Universal Robots PolyScope program: TCP Test 01.urp

Program TCP Test 01 (installation=default directory=/programs createdIn=5.9.1.1031110 lastSavedIn=5.9.1.1031110 robotSerialNumber=20195501059)
Calibrated DH parameters: a=[0.000146, -0.418764, -0.053981, 0.000058, -0.000023, 0]; d=[0.162545, 37.319448, -206.067439, 168.881546, 0.09955, 0.099464]; alpha=[1.57004, -0.001979, 0.002304, 1.570607, -1.57066, 0]; deltaTheta=[0, -0.174616, -1.258233, 1.432844, -0.000001, 0]
BeforeStart
  URCap Gripper Activate (Robotiq_Grippers, Robotiq Inc.) dataModel(ResetAndActivateKey=false)
  URCap Gripper (Robotiq_Grippers, Robotiq Inc.) dataModel(position=100.0, force=100.0, speed=100.0, positionInDouble=100.0, forceInDouble=100.0, speedInDouble=100.0, slaveIds=[9], blocking=true)
Robot Program (runOnlyOnce=true)
  '2F85 Tool vertical above box'
  MoveJ speed 60 deg/s, acceleration 80 deg/s^2 (useActiveTCP=false) tcp=TCP_2F85; feature=Base
    Waypoint hover: TCP in base x=299.991 y=-399.96 z=49.999 mm, rx=0.0001 ry=0.0001 rz=0 rad; joints [111.356, -78.636, 119.104, -130.453, 270.052, 201.393] deg; TCP offset x=0 y=0 z=175 mm, rx=3.1416 ry=0 rz=0 rad
    Waypoint on_target: TCP in base x=300.002 y=-399.956 z=0.996 mm, rx=0.0001 ry=0 rz=0 rad; joints [111.352, -73.264, 121.787, -138.509, 270.053, 201.401] deg; TCP offset x=0 y=0 z=175 mm, rx=3.1416 ry=0 rz=0 rad
  MoveJ speed 60 deg/s, acceleration 80 deg/s^2 (useActiveTCP=false) tcp=TCP_Mono; feature=Base
    Waypoint on_target: TCP in base x=300.002 y=-399.956 z=0.996 mm, rx=0.0001 ry=0 rz=0 rad; joints [111.352, -73.264, 121.787, -138.509, 270.053, 201.401] deg
  MoveJ speed 60 deg/s, acceleration 80 deg/s^2 (useActiveTCP=false) tcp=TCP_Color; feature=Base
    Waypoint on_target: TCP in base x=300.002 y=-399.956 z=0.996 mm, rx=0.0001 ry=0 rz=0 rad; joints [111.352, -73.264, 121.787, -138.509, 270.053, 201.401] deg
  MoveJ speed 60 deg/s, acceleration 80 deg/s^2 (useActiveTCP=false) tcp=TCP_Wenglor; feature=Base
    Waypoint on_target: TCP in base x=300.002 y=-399.956 z=0.996 mm, rx=0.0001 ry=0 rz=0 rad; joints [111.352, -73.264, 121.787, -138.509, 270.053, 201.401] deg
  MoveJ speed 60 deg/s, acceleration 80 deg/s^2 (useActiveTCP=false) tcp=TCP_2F85; feature=Base
    Waypoint hover: TCP in base x=299.991 y=-399.96 z=49.999 mm, rx=0.0001 ry=0.0001 rz=0 rad; joints [111.356, -78.636, 119.104, -130.453, 270.052, 201.393] deg; TCP offset x=0 y=0 z=175 mm, rx=3.1416 ry=0 rz=0 rad
